{attribute addProperty BoxType "EL2596-0000-0017"}
{attribute addProperty Id "EnableBIT10.1251OutputBIT10.1252Input_trigger_enableBIT10.1254Output_trigger_enableBIT10.1255ResetBIT10.1258"}
{attribute addProperty CRC "1254697747"}
{attribute addProperty SizeInBites "16"}
{attribute addProperty SizeInBytes "2"}
TYPE Control_4AC92B13 :
STRUCT
	{attribute addProperty Name "Enable"}
	Enable : BIT;
	{attribute addProperty Name "Output"}
	Output : BIT;
	{attribute 'hide'}
	reserve_1 : BIT;
	{attribute addProperty Name "Input_trigger_enable"}
	Input_trigger_enable : BIT;
	{attribute addProperty Name "Output_trigger_enable"}
	Output_trigger_enable : BIT;
	{attribute 'hide'}
	reserve_2_BIT_0 : BIT;
	{attribute 'hide'}
	reserve_2_BIT_1 : BIT;
	{attribute addProperty Name "Reset"}
	Reset : BIT;
	{attribute 'hide'}
	reserve_3 : BYTE;
END_STRUCT
END_TYPE

(* stored: Version 1.2.0.0, ProductVersion 3.1.4024.9
   DUT Control_4AC92B13: Id {ebe2c56a-d397-40b5-9ddb-27aa2521fb3a} *)
